FUNCTION_BLOCK FB_MovingAverage_Test EXTENDS TcUnit.FB_TestSuite


calculationShouldBeReadyWhenTimePassed();
calculationShouldNotBeReadyBeforeTimePassed();
movingAverageOfThreePlusTwoPlusOneShouldBeTwo();
resetMethodCallShouldResetValue();

METHOD calculationShouldBeReadyWhenTimePassed : BOOL
VAR
	movingAverage : FB_MovingAverage;
END_VAR

TEST('calculationShouldBeReadyWhenTimePassed');
movingAverage.startCalculation(TRUE,0, 3,1, T#3S);
AssertEquals_BOOL(Expected := TRUE, Actual :=  movingAverage.ready, Message := 'Moving average calculation not ready after time passed');
TEST_FINISHED();
END_METHOD

METHOD calculationShouldNotBeReadyBeforeTimePassed : BOOL
VAR
	movingAverage : FB_MovingAverage;
END_VAR

TEST('calculationShouldNotBeReadyBeforeTimePassed');
movingAverage.startCalculation(TRUE, 0, 1,1, T#0S);
AssertEquals_BOOL(Expected := FALSE, Actual :=  movingAverage.ready, Message := 'Moving average calculation ready before time passed');
TEST_FINISHED();
END_METHOD

METHOD movingAverageOfThreePlusTwoPlusOneShouldBeTwo
VAR
	movingAverage : FB_MovingAverage;
END_VAR

TEST('movingAverageOfThreePlusTwoPlusOneShouldBeTwo');
movingAverage.startCalculation(TRUE, 3, 3, 1, T#1S);
movingAverage.startCalculation(TRUE, 2, 3, 1, T#1S);
movingAverage.startCalculation(TRUE, 1, 3, 1, T#1S);
movingAverage.startCalculation(TRUE, 0, 3, 1, T#1S);
AssertEquals_REAL(Expected := 2, Actual := movingAverage.value, 0, Message := 'Moving average calculation not equal to two!');
TEST_FINISHED();
END_METHOD

METHOD resetMethodCallShouldResetValue
VAR
	movingAverage : FB_MovingAverage;
END_VAR

TEST('resetMethodCallShouldResetValue');
movingAverage.startCalculation(start := TRUE, measurement := 50, intervalS := 1, windowS := 3, dtime := T#3S);
movingAverage.reset();
AssertEquals_REAL(0, movingAverage.value, 0, 'Reset did not reset value!'); 
TEST_FINISHED();
END_METHOD

END_FUNCTION_BLOCK

(* stored: Version 1.1.0.1, ProductVersion 3.1.4024.9
   POU FB_MovingAverage_Test: Id {37b413a4-f223-4570-9474-bb8c477d7df3}, SpecialFunc None
   Method calculationShouldBeReadyWhenTimePassed: Id {6eb0e18c-3c4c-41df-9aec-1ae6efb07c6f}
   Method calculationShouldNotBeReadyBeforeTimePassed: Id {0d5beb96-f79e-4026-9737-489b3f97c409}
   Method movingAverageOfThreePlusTwoPlusOneShouldBeTwo: Id {6fbf797b-777c-48ee-9f5a-eb7f5971efd2}
   Method resetMethodCallShouldResetValue: Id {a1bce5bc-4342-4398-8196-3d4fc31f55c7} *)
